FUNCTION_BLOCK logiBUS_PI_IDA (* Composite FB for double word input data *)
  (* Standard: 61499-2; Description: Copyright (c) 2026 HR Agrartechnik GmbH This program and the accompanying materials are made available under the terms of the Eclipse Public License 2.0 which is available at https://www.eclipse.org/legal/epl-2.0/ SPDX-License-Identifier: EPL-2.0 if ImpulseDelta = 0, then TimeDelta cannot be 0. set TimeDelta to 16#FFFFFFFF to deactivate cyclic processing, and onyl indicate Changes in Value. *)
  (* Version 1.0, 2026-02-23, Franz Höpfinger, HR Agrartechnik GmbH *)
  PACKAGE logiBUS::io::PI;
  IMPORT eclipse4diac::core::TypeHash;
  IMPORT logiBUS::io::PI::logiBUS_PI::Invalid;
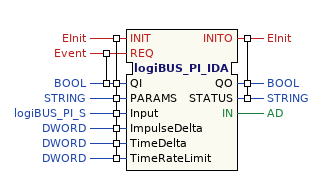
  EVENT_INPUT
    INIT : EInit WITH QI, PARAMS, Input, ImpulseDelta, TimeDelta, TimeRateLimit; (* Service Initialization *)
    REQ WITH QI; (* Service Request *)
  END_EVENT
  EVENT_OUTPUT
    INITO : EInit WITH QO, STATUS; (* Initialization Confirm *)
  END_EVENT
  VAR_INPUT
    QI : BOOL; (* Event Input Qualifier *)
    PARAMS : STRING; (* Service Parameters *)
    Input : logiBUS::io::PI::logiBUS_PI_S := Invalid; (* Identify the Input Input_I1..I8 *)
    ImpulseDelta : DWORD; (* After How many Impulses an IND *)
    TimeDelta : DWORD := 250; (* After How many ms an IND *)
    TimeRateLimit : DWORD := 100; (* Maximum 1 IND in how many ms. (< delta) *)
  END_VAR
  VAR_OUTPUT
    QO : BOOL; (* Event Output Qualifier *)
    STATUS : STRING; (* Service Status *)
  END_VAR
  PLUGS
    IN : adapter::types::unidirectional::AD; (* Input data from resource *)
  END_PLUGS
  FBS
    PI : logiBUS::io::PI::logiBUS_PI_ID;
  END_FBS
  EVENT_CONNECTIONS
    INIT TO PI.INIT;
    PI.INITO TO INITO;
    PI.IND TO IN.E1;
    PI.CNF TO IN.E1;
    REQ TO PI.REQ;
  END_CONNECTIONS
  DATA_CONNECTIONS
    PI.IN TO IN.D1;
    QI TO PI.QI;
    PARAMS TO PI.PARAMS;
    PI.QO TO QO;
    PI.STATUS TO STATUS;
    Input TO PI.Input;
    ImpulseDelta TO PI.ImpulseDelta;
    TimeDelta TO PI.TimeDelta;
    TimeRateLimit TO PI.TimeRateLimit;
  END_CONNECTIONS
END_FUNCTION_BLOCK
